LIN {X 0,Y 60.605,Z 418.461,A -85,B 0,C 180,E1 -30804.75,E2 -30804.75} C_VEL
LIN {X 0,Y 56.521,Z 422.655,A -85,B 0,C 180,E1 -30805.679,E2 -30805.679} C_VEL
LIN {X 0,Y 45.748,Z 431.459,A -85,B 0,C 180,E1 -30805.46,E2 -30805.46} C_VEL
LIN {X 0,Y 39.288,Z 436.041,A -85,B 0,C 180,E1 -30806.118,E2 -30806.118} C_VEL
LIN {X 0,Y 36.151,Z 438.173,A -85,B 0,C 180,E1 -30807.638,E2 -30807.638} C_VEL
LIN {X 0,Y 26.416,Z 444.355,A -85,B 0,C 180,E1 -30817.1,E2 -30817.1} C_VEL
LIN {X 0,Y 18.209,Z 449.039,A -85,B 0,C 180,E1 -30834.68,E2 -30834.68} C_VEL
LIN {X 0,Y 13.118,Z 452.656,A -85,B 0,C 180,E1 -30870.058,E2 -30870.058} C_VEL
LIN {X 0,Y 13.689,Z 454.507,A -85,B 0,C 180,E1 -30900.953,E2 -30900.953} C_VEL
LIN {X 0,Y 22.822,Z 456.912,A -85,B 0,C 180,E1 -30937.567,E2 -30937.567} C_VEL
LIN {X 0,Y 29.16,Z 457.53,A -85,B 0,C 180,E1 -30946.052,E2 -30946.052} C_VEL
LIN {X 0,Y 42.32,Z 457.444,A -85,B 0,C 180,E1 -30955.289,E2 -30955.289} C_VEL
LIN {X 0,Y 55.538,Z 455.876,A -85,B 0,C 180,E1 -30959.999,E2 -30959.999} C_VEL
LIN {X 0,Y 66.838,Z 453.338,A -85,B 0,C 180,E1 -30962.54,E2 -30962.54} C_VEL
LIN {X 0,Y 70.396,Z 452.283,A -85,B 0,C 180,E1 -30963.198,E2 -30963.198} C_VEL
LIN {X 0,Y 70.514,Z 452.314,A -85,B 0,C 180,E1 -30964.606,E2 -30964.606} C_VEL
LIN {X 0,Y 56.686,Z 455.939,A -85,B 0,C 180,E1 -30967.256,E2 -30967.256} C_VEL
LIN {X 0,Y 49.839,Z 457.143,A -85,B 0,C 180,E1 -30969.156,E2 -30969.156} C_VEL
LIN {X 0,Y 36.383,Z 458.329,A -85,B 0,C 180,E1 -30974.963,E2 -30974.963} C_VEL
LIN {X 0,Y 29.89,Z 458.361,A -85,B 0,C 180,E1 -30979.805,E2 -30979.805} C_VEL
LIN {X 0,Y 23.801,Z 458.025,A -85,B 0,C 180,E1 -30987.586,E2 -30987.586} C_VEL
LIN {X 0,Y 14.509,Z 456.115,A -85,B 0,C 180,E1 -31020.971,E2 -31020.971} C_VEL
LIN {X 0,Y 13.201,Z 454.549,A -85,B 0,C 180,E1 -31049.943,E2 -31049.943} C_VEL
LIN {X 0,Y 16.073,Z 451.235,A -85,B 0,C 180,E1 -31090.92,E2 -31090.92} C_VEL
LIN {X 0,Y 23.636,Z 446.806,A -85,B 0,C 180,E1 -31113.046,E2 -31113.046} C_VEL
LIN {X 0,Y 32.965,Z 441.169,A -85,B 0,C 180,E1 -31123.513,E2 -31123.513} C_VEL
LIN {X 0,Y 42.849,Z 434.081,A -85,B 0,C 180,E1 -31129.643,E2 -31129.643} C_VEL
LIN {X 0,Y 53.078,Z 425.225,A -85,B 0,C 180,E1 -31133.083,E2 -31133.083} C_VEL
LIN {X 0,Y 61.678,Z 416.099,A -85,B 0,C 180,E1 -31135.353,E2 -31135.353} C_VEL
LIN {X 0,Y 69.499,Z 406.088,A -85,B 0,C 180,E1 -31136.668,E2 -31136.668} C_VEL
LIN {X 0,Y 76.476,Z 394.946,A -85,B 0,C 180,E1 -31137.598,E2 -31137.598} C_VEL
LIN {X 0,Y 82.155,Z 383.414,A -85,B 0,C 180,E1 -31138.301,E2 -31138.301} C_VEL
LIN {X 0,Y 86.783,Z 371.031,A -85,B 0,C 180,E1 -31138.775,E2 -31138.775} C_VEL
LIN {X 0,Y 90.148,Z 357.801,A -85,B 0,C 180,E1 -31139.148,E2 -31139.148} C_VEL
LIN {X 0,Y 91.905,Z 346.427,A -85,B 0,C 180,E1 -31139.436,E2 -31139.436} C_VEL
LIN {X 0,Y 91.676,Z 344.487,A -85,B 0,C 180,E1 -31143.236,E2 -31143.236} C_VEL
LIN {X 0,Y 91.633,Z 344.144,A -85,B 0,C 180,E1 -31145.252,E2 -31145.252} C_VEL
LIN {X 0,Y 91.721,Z 345.464,A -85,B 0,C 180,E1 -31150.208,E2 -31150.208} C_VEL
LIN {X 0,Y 91.858,Z 346.545,A -85,B 0,C 180,E1 -31152.086,E2 -31152.086} C_VEL
LIN {X 0,Y 89.523,Z 360.208,A -85,B 0,C 180,E1 -31152.481,E2 -31152.481} C_VEL
LIN {X 0,Y 85.807,Z 373.355,A -85,B 0,C 180,E1 -31153.065,E2 -31153.065} C_VEL
LIN {X 0,Y 81.328,Z 384.734,A -85,B 0,C 180,E1 -31153.84,E2 -31153.84} C_VEL
LIN {X 0,Y 75.412,Z 396.214,A -85,B 0,C 180,E1 -31154.844,E2 -31154.844} C_VEL
LIN {X 0,Y 67.709,Z 407.907,A -85,B 0,C 180,E1 -31156.295,E2 -31156.295} C_VEL
LIN {X 0,Y 60.824,Z 416.395,A -85,B 0,C 180,E1 -31157.647,E2 -31157.647} C_VEL
LIN {X 0,Y 52.359,Z 425.167,A -85,B 0,C 180,E1 -31160.075,E2 -31160.075} C_VEL
LIN {X 0,Y 43.984,Z 432.411,A -85,B 0,C 180,E1 -31163.31,E2 -31163.31} C_VEL
LIN {X 0,Y 36.151,Z 438.173,A -85,B 0,C 180,E1 -31167.638,E2 -31167.638} C_VEL
LIN {X 0,Y 31.341,Z 441.245,A -85,B 0,C 180,E1 -31170.246,E2 -31170.246} C_VEL
LIN {X 0,Y 22.613,Z 445.789,A -85,B 0,C 180,E1 -31172.884,E2 -31172.884} C_VEL
LIN {X 0,Y 13.538,Z 449.603,A -85,B 0,C 180,E1 -31178.355,E2 -31178.355} C_VEL
LIN {X 0,Y 8.599,Z 451.538,A -85,B 0,C 180,E1 -31192.825,E2 -31192.825} C_VEL
LIN {X 0,Y 8.347,Z 454.988,A -85,B 0,C 180,E1 -31287.507,E2 -31287.507} C_VEL
LIN {X 0,Y 14.382,Z 456.359,A -85,B 0,C 180,E1 -31308.006,E2 -31308.006} C_VEL
LIN {X 0,Y 27.155,Z 457.834,A -85,B 0,C 180,E1 -31319.999,E2 -31319.999} C_VEL
LIN {X 0,Y 35.208,Z 458.006,A -85,B 0,C 180,E1 -31323.307,E2 -31323.307} C_VEL
LIN {X 0,Y 35.223,Z 458.016,A -85,B 0,C 180,E1 -31323.69,E2 -31323.69} C_VEL
LIN {X 0,Y 28.282,Z 458.017,A -85,B 0,C 180,E1 -31326.093,E2 -31326.093} C_VEL
LIN {X 0,Y 21.451,Z 457.632,A -85,B 0,C 180,E1 -31330.451,E2 -31330.451} C_VEL
LIN {X 0,Y 8.981,Z 455.649,A -85,B 0,C 180,E1 -31358.374,E2 -31358.374} C_VEL
LIN {X 0,Y 6.112,Z 454.053,A -85,B 0,C 180,E1 -31409.876,E2 -31409.876} C_VEL
LIN {X 0,Y 11.66,Z 450.669,A -85,B 0,C 180,E1 -31474.544,E2 -31474.544} C_VEL
LIN {X 0,Y 21.368,Z 446.167,A -85,B 0,C 180,E1 -31490.4,E2 -31490.4} C_VEL
LIN {X 0,Y 31.685,Z 440.451,A -85,B 0,C 180,E1 -31496.043,E2 -31496.043} C_VEL
LIN {X 0,Y 42.153,Z 433.225,A -85,B 0,C 180,E1 -31499.342,E2 -31499.342} C_VEL
LIN {X 0,Y 52.697,Z 424.271,A -85,B 0,C 180,E1 -31500.826,E2 -31500.826} C_VEL
LIN {X 0,Y 61.515,Z 415.012,A -85,B 0,C 180,E1 -31502.057,E2 -31502.057} C_VEL
LIN {X 0,Y 69.449,Z 404.793,A -85,B 0,C 180,E1 -31502.521,E2 -31502.521} C_VEL
LIN {X 0,Y 76.51,Z 393.402,A -85,B 0,C 180,E1 -31502.952,E2 -31502.952} C_VEL
LIN {X 0,Y 81.814,Z 382.55,A -85,B 0,C 180,E1 -31503.291,E2 -31503.291} C_VEL
LIN {X 0,Y 86.33,Z 370.462,A -85,B 0,C 180,E1 -31503.468,E2 -31503.468} C_VEL
LIN {X 0,Y 89.679,Z 357.327,A -85,B 0,C 180,E1 -31503.65,E2 -31503.65} C_VEL
LIN {X 0,Y 90.705,Z 351.469,A -85,B 0,C 180,E1 -31503.755,E2 -31503.755} C_VEL
LIN {X 0,Y 90.652,Z 351.439,A -85,B 0,C 180,E1 -31506.121,E2 -31506.121} C_VEL
LIN {X 0,Y 90.642,Z 351.789,A -85,B 0,C 180,E1 -31507.689,E2 -31507.689} C_VEL
LIN {X 0,Y 87.922,Z 364.791,A -85,B 0,C 180,E1 -31508.029,E2 -31508.029} C_VEL
LIN {X 0,Y 83.72,Z 377.67,A -85,B 0,C 180,E1 -31508.514,E2 -31508.514} C_VEL
LIN {X 0,Y 78.274,Z 389.889,A -85,B 0,C 180,E1 -31509.109,E2 -31509.109} C_VEL
LIN {X 0,Y 72.172,Z 400.509,A -85,B 0,C 180,E1 -31509.709,E2 -31509.709} C_VEL
LIN {X 0,Y 65.173,Z 410.317,A -85,B 0,C 180,E1 -31510.357,E2 -31510.357} C_VEL
LIN {X 0,Y 57.321,Z 419.36,A -85,B 0,C 180,E1 -31511.321,E2 -31511.321} C_VEL
LIN {X 0,Y 46.901,Z 429.125,A -85,B 0,C 180,E1 -31513.185,E2 -31513.185} C_VEL
LIN {X 0,Y 36.489,Z 436.97,A -85,B 0,C 180,E1 -31515.724,E2 -31515.724} C_VEL
LIN {X 0,Y 26.227,Z 443.222,A -85,B 0,C 180,E1 -31520.398,E2 -31520.398} C_VEL
LIN {X 0,Y 16.221,Z 448.213,A -85,B 0,C 180,E1 -31530.044,E2 -31530.044} C_VEL
LIN {X 0,Y 8.599,Z 451.538,A -85,B 0,C 180,E1 -31552.825,E2 -31552.825} C_VEL
LIN {X 0,Y 7.625,Z 453.446,A -85,B 0,C 180,E1 -31559.956,E2 -31559.956} C_VEL
LIN {X 0,Y 7.625,Z 600,A -85,B 0,C 180,E1 -31559.956,E2 -31559.956} C_VEL
LIN {X 0,Y 7.625,Z 600,A -85,B 0,C 180,E1 -31559.956,E2 -31559.956}

QRS_NEXT_CUT()

QRS_NEXT()
QRS_HOME()

END
